Universal Robots PolyScope program: bearing_plate_positioning2.urp

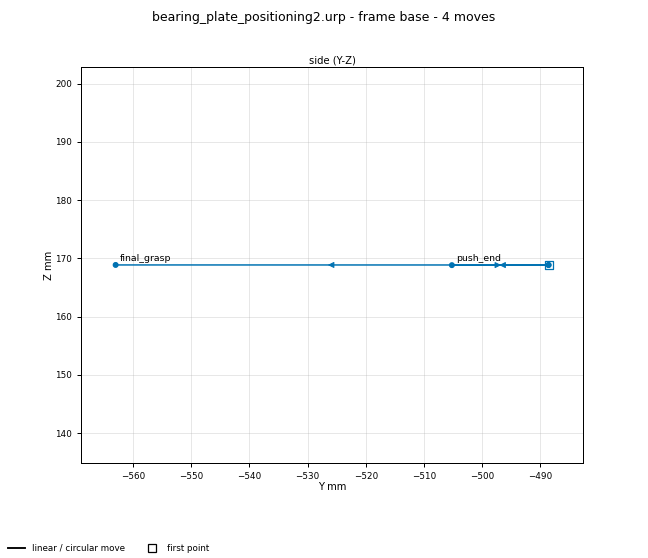
[picture p0: tool path of bearing_plate_positioning2.urp in frame base, 4 of 5 moves have a stored position in this frame; points joined in program order, loops and branches not executed]
Program bearing_plate_positioning2 (installation=default directory=/programs/wrs2020 createdIn=5.9.1.1031110 lastSavedIn=5.9.1.1031110 robotSerialNumber=20205500180)
Calibrated DH parameters: a=[0, -0.425, -0.3922, 0, 0, 0]; d=[0.1625, 0, 0, 0.1333, 0.0997, 0.0996]; alpha=[1.570796, 0, 0, 1.570796, -1.570796, 0]; deltaTheta=[0, 0, 0, 0, 0, 0]
Robot Program (runOnlyOnce=true)
  URCap Gripper (Robotiq_Grippers, Robotiq Inc.) dataModel(position=51.76470588235294, force=100.0, speed=100.0, positionInDouble=51.76470588235294, forceInDouble=100.0, speedInDouble=100.0, slaveIds=[9], blocking=true)
  MoveJ speed 60 deg/s, acceleration 80 deg/s^2 (useActiveTCP=true) feature=Base
    currentpose := get_actual_tcp_pose()get_actual_joint_positions()
    Waypoint Waypoint (Variable): variable=currentpose
  MoveL speed 250 mm/s, acceleration 1200 mm/s^2 (useActiveTCP=false) tcp=gripper_140_tip; feature=Base
    Waypoint before_push: TCP in base x=91.011 y=-488.607 z=168.87 mm, rx=2.4445 ry=-0.0026 rz=0.0045 rad; joints [81.025, -109.238, 142.198, -162.536, -84.106, 173.271] deg; TCP offset x=0 y=0 z=220 mm, rx=0 ry=0 rz=0 rad
  URCap Gripper (Robotiq_Grippers, Robotiq Inc.) dataModel(position=100.0, force=100.0, speed=100.0, positionInDouble=100.0, forceInDouble=100.0, speedInDouble=100.0, slaveIds=[9], blocking=true)
  MoveL speed 250 mm/s, acceleration 1200 mm/s^2 (useActiveTCP=false) tcp=gripper_140_tip; feature=Base
    Waypoint push_end: motionParameters(jointSpeed=1.047198 jointAcceleration=1.396263 cartesianSpeed=0.05 cartesianAcceleration=0.02); TCP in base x=90.982 y=-505.209 z=168.841 mm, rx=2.4446 ry=-0.0028 rz=0.0045 rad; joints [81.547, -106.058, 140.283, -163.838, -84.44, 173.682] deg
    Waypoint before_push: motionParameters(jointSpeed=1.047198 jointAcceleration=1.396263 cartesianSpeed=0.25 cartesianAcceleration=0.5); TCP in base x=91.011 y=-488.607 z=168.87 mm, rx=2.4445 ry=-0.0026 rz=0.0045 rad; joints [81.025, -109.238, 142.198, -162.536, -84.106, 173.271] deg
  URCap Gripper (Robotiq_Grippers, Robotiq Inc.) dataModel(position=51.76470588235294, force=100.0, speed=100.0, positionInDouble=51.76470588235294, forceInDouble=100.0, speedInDouble=100.0, slaveIds=[9], blocking=true)
  MoveL speed 500 mm/s, acceleration 800 mm/s^2 (useActiveTCP=false) tcp=gripper_140_tip; feature=Base
    SuppressedNode
      Waypoint Waypoint_2: TCP in base x=89.229 y=-495.285 z=194.846 mm, rx=0.0168 ry=3.034 rz=-0.7765 rad; joints [82.081, -107.449, 128.407, -139.394, -85.816, -6.224] deg
    Waypoint final_grasp: TCP in base x=90.974 y=-562.948 z=168.878 mm, rx=2.3752 ry=-0.0026 rz=0.0045 rad; joints [82.613, -95.841, 136.395, -174.212, -84.741, 174.847] deg
  URCap Gripper (Robotiq_Grippers, Robotiq Inc.) dataModel(position=100.0, force=0.0, speed=0.0, positionInDouble=100.0, forceInDouble=0.0, speedInDouble=0.0, slaveIds=[9], blocking=true)
  URCap Gripper (Robotiq_Grippers, Robotiq Inc.) dataModel(position=84.70588235294117, force=100.0, speed=0.0, positionInDouble=84.70588235294117, forceInDouble=100.0, speedInDouble=0.0, slaveIds=[9], blocking=true)
